// TIA Portal V15.1 export
// export: Created 2024-06-21T08:41:25.9680752Z, ExportSetting WithDefaults, DisplayName Totally Integrated Automation Portal, DisplayVersion V15.1 Update 5, DisplayName TIA Portal Openness, DisplayVersion V15.1 Update 5, DisplayName SINAMICS Startdrive Advanced, DisplayVersion V15.1, DisplayName G130, G150, S120, S150, SINAMICS MV, S210, DisplayVersion V15.1, DisplayName G110M, G120, G120C, G120D, G120P, DisplayVersion V15.1, DisplayName STEP 7 Professional, DisplayVersion V15.1 Update 5, DisplayName STEP 7 Safety, DisplayVersion V15.1, DisplayName WinCC Professional, DisplayVersion V15.1 Update 5, DisplayName SIMATIC Visualization Architect, DisplayVersion V15.1
FUNCTION "209000NCP01EnableAlarms" : Void   // FC198, FBD
TITLE = 209000NCP01EnableAlarms
{ S7_Optimized_Access := 'TRUE' }
VERSION : 0.1
// stored: AutoNumber false, IsIECCheckEnabled false, SetENOAutomatically False, UDAEnableTagReadback false
BEGIN

REGION Network 1: **** --------------------- General --------------------- ****
END_REGION

REGION Network 2: **** 2.1 - Enable Alarms **** General Switch - 209000AE02-JW210
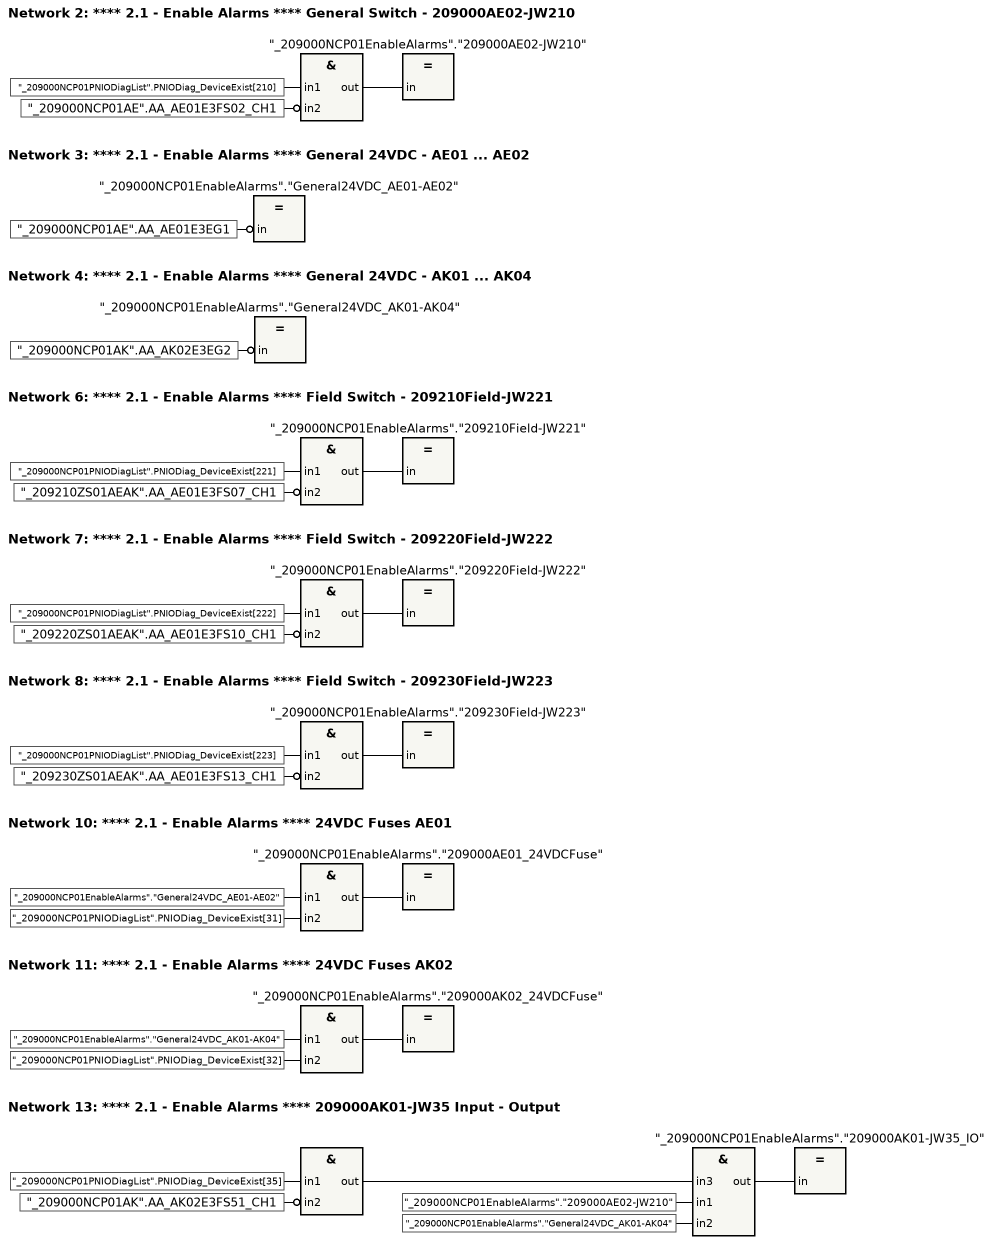
   "_209000NCP01EnableAlarms"."209000AE02-JW210" := "_209000NCP01PNIODiagList".PNIODiag_DeviceExist[210] AND NOT "_209000NCP01AE".AA_AE01E3FS02_CH1;
END_REGION

REGION Network 3: **** 2.1 - Enable Alarms **** General 24VDC - AE01 ... AE02
   "_209000NCP01EnableAlarms"."General24VDC_AE01-AE02" := NOT "_209000NCP01AE".AA_AE01E3EG1;
END_REGION

REGION Network 4: **** 2.1 - Enable Alarms **** General 24VDC - AK01 ... AK04
   "_209000NCP01EnableAlarms"."General24VDC_AK01-AK04" := NOT "_209000NCP01AK".AA_AK02E3EG2;
END_REGION

REGION Network 5: **** --------------------- Field Switch --------------------- ****
END_REGION

REGION Network 6: **** 2.1 - Enable Alarms **** Field Switch - 209210Field-JW221
   "_209000NCP01EnableAlarms"."209210Field-JW221" := "_209000NCP01PNIODiagList".PNIODiag_DeviceExist[221] AND NOT "_209210ZS01AEAK".AA_AE01E3FS07_CH1;
END_REGION

REGION Network 7: **** 2.1 - Enable Alarms **** Field Switch - 209220Field-JW222
   "_209000NCP01EnableAlarms"."209220Field-JW222" := "_209000NCP01PNIODiagList".PNIODiag_DeviceExist[222] AND NOT "_209220ZS01AEAK".AA_AE01E3FS10_CH1;
END_REGION

REGION Network 8: **** 2.1 - Enable Alarms **** Field Switch - 209230Field-JW223
   "_209000NCP01EnableAlarms"."209230Field-JW223" := "_209000NCP01PNIODiagList".PNIODiag_DeviceExist[223] AND NOT "_209230ZS01AEAK".AA_AE01E3FS13_CH1;
END_REGION

REGION Network 9: **** --------------------- ETA Fuse --------------------- ****
END_REGION

REGION Network 10: **** 2.1 - Enable Alarms **** 24VDC Fuses AE01
   "_209000NCP01EnableAlarms"."209000AE01_24VDCFuse" := "_209000NCP01EnableAlarms"."General24VDC_AE01-AE02" AND "_209000NCP01PNIODiagList".PNIODiag_DeviceExist[31];
END_REGION

REGION Network 11: **** 2.1 - Enable Alarms **** 24VDC Fuses AK02
   "_209000NCP01EnableAlarms"."209000AK02_24VDCFuse" := "_209000NCP01EnableAlarms"."General24VDC_AK01-AK04" AND "_209000NCP01PNIODiagList".PNIODiag_DeviceExist[32];
END_REGION

REGION Network 12: **** --------------------- ET200sp I/O --------------------- ****
END_REGION

REGION Network 13: **** 2.1 - Enable Alarms **** 209000AK01-JW35 Input - Output
   "_209000NCP01EnableAlarms"."209000AK01-JW35_IO" := "_209000NCP01PNIODiagList".PNIODiag_DeviceExist[35] AND NOT "_209000NCP01AK".AA_AK02E3FS51_CH1 AND "_209000NCP01EnableAlarms"."209000AE02-JW210" AND "_209000NCP01EnableAlarms"."General24VDC_AK01-AK04";
END_REGION

REGION Network 14: **** 2.1 - Enable Alarms **** 209000AK01-JW35 Safety Input - Output
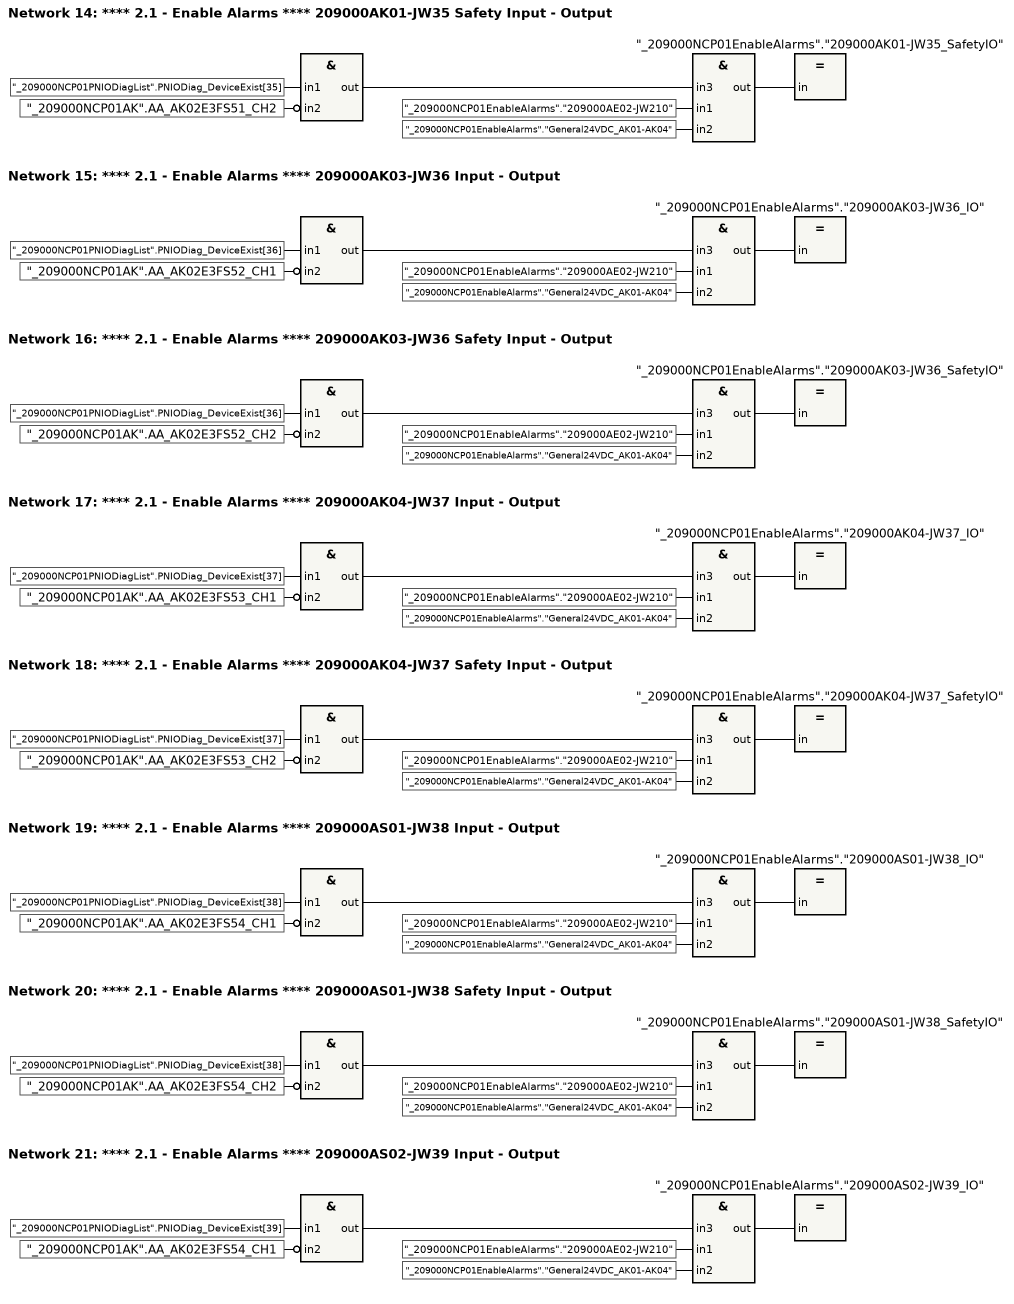
   "_209000NCP01EnableAlarms"."209000AK01-JW35_SafetyIO" := "_209000NCP01PNIODiagList".PNIODiag_DeviceExist[35] AND NOT "_209000NCP01AK".AA_AK02E3FS51_CH2 AND "_209000NCP01EnableAlarms"."209000AE02-JW210" AND "_209000NCP01EnableAlarms"."General24VDC_AK01-AK04";
END_REGION

REGION Network 15: **** 2.1 - Enable Alarms **** 209000AK03-JW36 Input - Output
   "_209000NCP01EnableAlarms"."209000AK03-JW36_IO" := "_209000NCP01PNIODiagList".PNIODiag_DeviceExist[36] AND NOT "_209000NCP01AK".AA_AK02E3FS52_CH1 AND "_209000NCP01EnableAlarms"."209000AE02-JW210" AND "_209000NCP01EnableAlarms"."General24VDC_AK01-AK04";
END_REGION

REGION Network 16: **** 2.1 - Enable Alarms **** 209000AK03-JW36 Safety Input - Output
   "_209000NCP01EnableAlarms"."209000AK03-JW36_SafetyIO" := "_209000NCP01PNIODiagList".PNIODiag_DeviceExist[36] AND NOT "_209000NCP01AK".AA_AK02E3FS52_CH2 AND "_209000NCP01EnableAlarms"."209000AE02-JW210" AND "_209000NCP01EnableAlarms"."General24VDC_AK01-AK04";
END_REGION

REGION Network 17: **** 2.1 - Enable Alarms **** 209000AK04-JW37 Input - Output
   "_209000NCP01EnableAlarms"."209000AK04-JW37_IO" := "_209000NCP01PNIODiagList".PNIODiag_DeviceExist[37] AND NOT "_209000NCP01AK".AA_AK02E3FS53_CH1 AND "_209000NCP01EnableAlarms"."209000AE02-JW210" AND "_209000NCP01EnableAlarms"."General24VDC_AK01-AK04";
END_REGION

REGION Network 18: **** 2.1 - Enable Alarms **** 209000AK04-JW37 Safety Input - Output
   "_209000NCP01EnableAlarms"."209000AK04-JW37_SafetyIO" := "_209000NCP01PNIODiagList".PNIODiag_DeviceExist[37] AND NOT "_209000NCP01AK".AA_AK02E3FS53_CH2 AND "_209000NCP01EnableAlarms"."209000AE02-JW210" AND "_209000NCP01EnableAlarms"."General24VDC_AK01-AK04";
END_REGION

REGION Network 19: **** 2.1 - Enable Alarms **** 209000AS01-JW38 Input - Output
   "_209000NCP01EnableAlarms"."209000AS01-JW38_IO" := "_209000NCP01PNIODiagList".PNIODiag_DeviceExist[38] AND NOT "_209000NCP01AK".AA_AK02E3FS54_CH1 AND "_209000NCP01EnableAlarms"."209000AE02-JW210" AND "_209000NCP01EnableAlarms"."General24VDC_AK01-AK04";
END_REGION

REGION Network 20: **** 2.1 - Enable Alarms **** 209000AS01-JW38 Safety Input - Output
   "_209000NCP01EnableAlarms"."209000AS01-JW38_SafetyIO" := "_209000NCP01PNIODiagList".PNIODiag_DeviceExist[38] AND NOT "_209000NCP01AK".AA_AK02E3FS54_CH2 AND "_209000NCP01EnableAlarms"."209000AE02-JW210" AND "_209000NCP01EnableAlarms"."General24VDC_AK01-AK04";
END_REGION

REGION Network 21: **** 2.1 - Enable Alarms **** 209000AS02-JW39 Input - Output
   "_209000NCP01EnableAlarms"."209000AS02-JW39_IO" := "_209000NCP01PNIODiagList".PNIODiag_DeviceExist[39] AND NOT "_209000NCP01AK".AA_AK02E3FS54_CH1 AND "_209000NCP01EnableAlarms"."209000AE02-JW210" AND "_209000NCP01EnableAlarms"."General24VDC_AK01-AK04";
END_REGION

REGION Network 22: **** 2.1 - Enable Alarms **** 209000AS02-JW39 Safety Input - Output
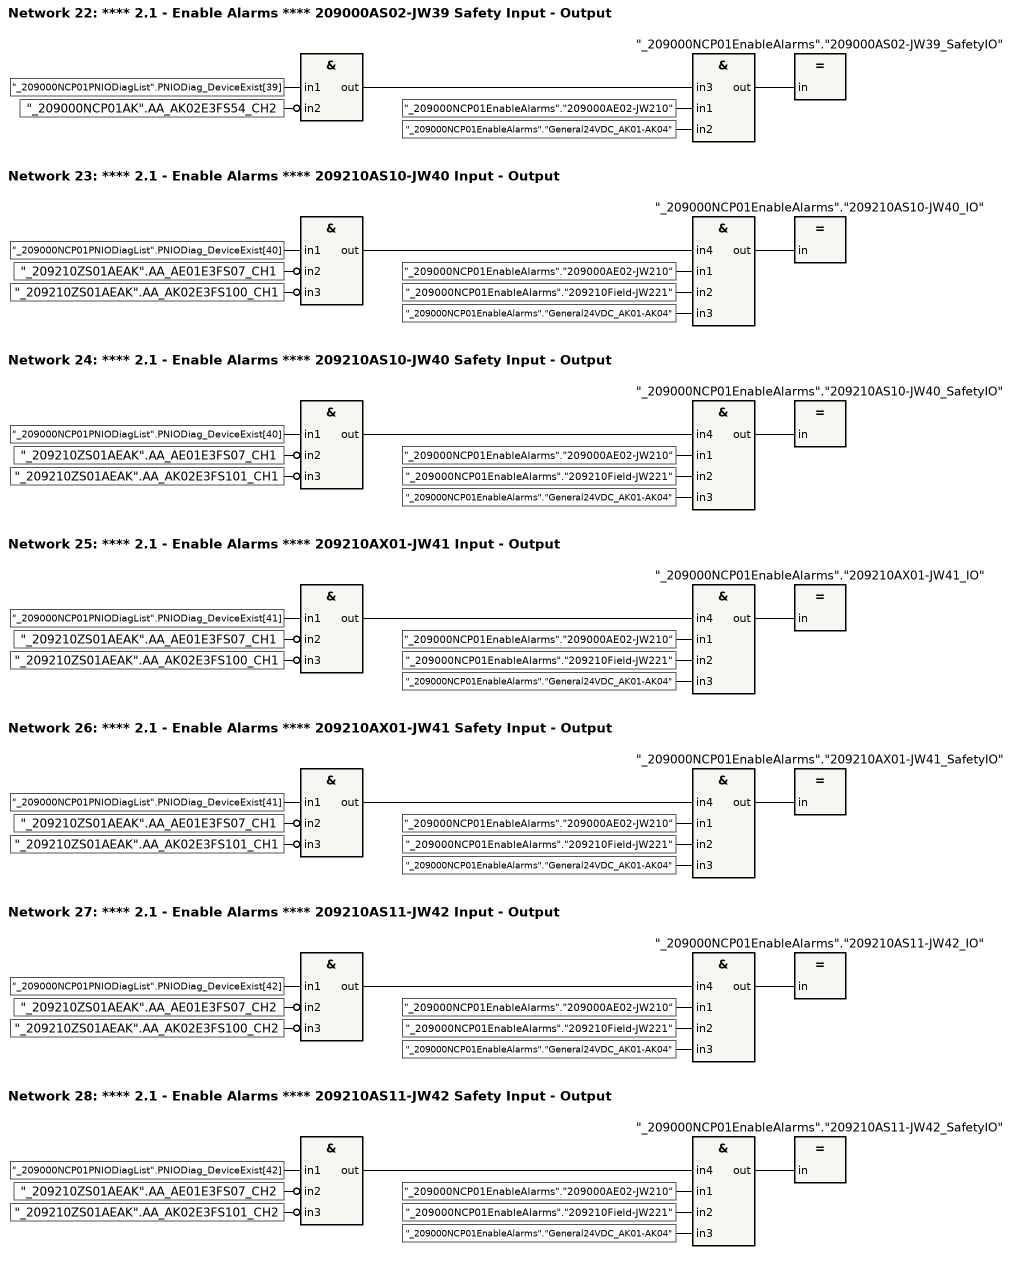
   "_209000NCP01EnableAlarms"."209000AS02-JW39_SafetyIO" := "_209000NCP01PNIODiagList".PNIODiag_DeviceExist[39] AND NOT "_209000NCP01AK".AA_AK02E3FS54_CH2 AND "_209000NCP01EnableAlarms"."209000AE02-JW210" AND "_209000NCP01EnableAlarms"."General24VDC_AK01-AK04";
END_REGION

REGION Network 23: **** 2.1 - Enable Alarms **** 209210AS10-JW40 Input - Output
   "_209000NCP01EnableAlarms"."209210AS10-JW40_IO" := "_209000NCP01PNIODiagList".PNIODiag_DeviceExist[40] AND NOT "_209210ZS01AEAK".AA_AE01E3FS07_CH1 AND NOT "_209210ZS01AEAK".AA_AK02E3FS100_CH1 AND "_209000NCP01EnableAlarms"."209000AE02-JW210" AND "_209000NCP01EnableAlarms"."209210Field-JW221" AND "_209000NCP01EnableAlarms"."General24VDC_AK01-AK04";
END_REGION

REGION Network 24: **** 2.1 - Enable Alarms **** 209210AS10-JW40 Safety Input - Output
   "_209000NCP01EnableAlarms"."209210AS10-JW40_SafetyIO" := "_209000NCP01PNIODiagList".PNIODiag_DeviceExist[40] AND NOT "_209210ZS01AEAK".AA_AE01E3FS07_CH1 AND NOT "_209210ZS01AEAK".AA_AK02E3FS101_CH1 AND "_209000NCP01EnableAlarms"."209000AE02-JW210" AND "_209000NCP01EnableAlarms"."209210Field-JW221" AND "_209000NCP01EnableAlarms"."General24VDC_AK01-AK04";
END_REGION

REGION Network 25: **** 2.1 - Enable Alarms **** 209210AX01-JW41 Input - Output
   "_209000NCP01EnableAlarms"."209210AX01-JW41_IO" := "_209000NCP01PNIODiagList".PNIODiag_DeviceExist[41] AND NOT "_209210ZS01AEAK".AA_AE01E3FS07_CH1 AND NOT "_209210ZS01AEAK".AA_AK02E3FS100_CH1 AND "_209000NCP01EnableAlarms"."209000AE02-JW210" AND "_209000NCP01EnableAlarms"."209210Field-JW221" AND "_209000NCP01EnableAlarms"."General24VDC_AK01-AK04";
END_REGION

REGION Network 26: **** 2.1 - Enable Alarms **** 209210AX01-JW41 Safety Input - Output
   "_209000NCP01EnableAlarms"."209210AX01-JW41_SafetyIO" := "_209000NCP01PNIODiagList".PNIODiag_DeviceExist[41] AND NOT "_209210ZS01AEAK".AA_AE01E3FS07_CH1 AND NOT "_209210ZS01AEAK".AA_AK02E3FS101_CH1 AND "_209000NCP01EnableAlarms"."209000AE02-JW210" AND "_209000NCP01EnableAlarms"."209210Field-JW221" AND "_209000NCP01EnableAlarms"."General24VDC_AK01-AK04";
END_REGION

REGION Network 27: **** 2.1 - Enable Alarms **** 209210AS11-JW42 Input - Output
   "_209000NCP01EnableAlarms"."209210AS11-JW42_IO" := "_209000NCP01PNIODiagList".PNIODiag_DeviceExist[42] AND NOT "_209210ZS01AEAK".AA_AE01E3FS07_CH2 AND NOT "_209210ZS01AEAK".AA_AK02E3FS100_CH2 AND "_209000NCP01EnableAlarms"."209000AE02-JW210" AND "_209000NCP01EnableAlarms"."209210Field-JW221" AND "_209000NCP01EnableAlarms"."General24VDC_AK01-AK04";
END_REGION

REGION Network 28: **** 2.1 - Enable Alarms **** 209210AS11-JW42 Safety Input - Output
   "_209000NCP01EnableAlarms"."209210AS11-JW42_SafetyIO" := "_209000NCP01PNIODiagList".PNIODiag_DeviceExist[42] AND NOT "_209210ZS01AEAK".AA_AE01E3FS07_CH2 AND NOT "_209210ZS01AEAK".AA_AK02E3FS101_CH2 AND "_209000NCP01EnableAlarms"."209000AE02-JW210" AND "_209000NCP01EnableAlarms"."209210Field-JW221" AND "_209000NCP01EnableAlarms"."General24VDC_AK01-AK04";
END_REGION

REGION Network 29: **** 2.1 - Enable Alarms **** 209210AX02-JW43 Input - Output
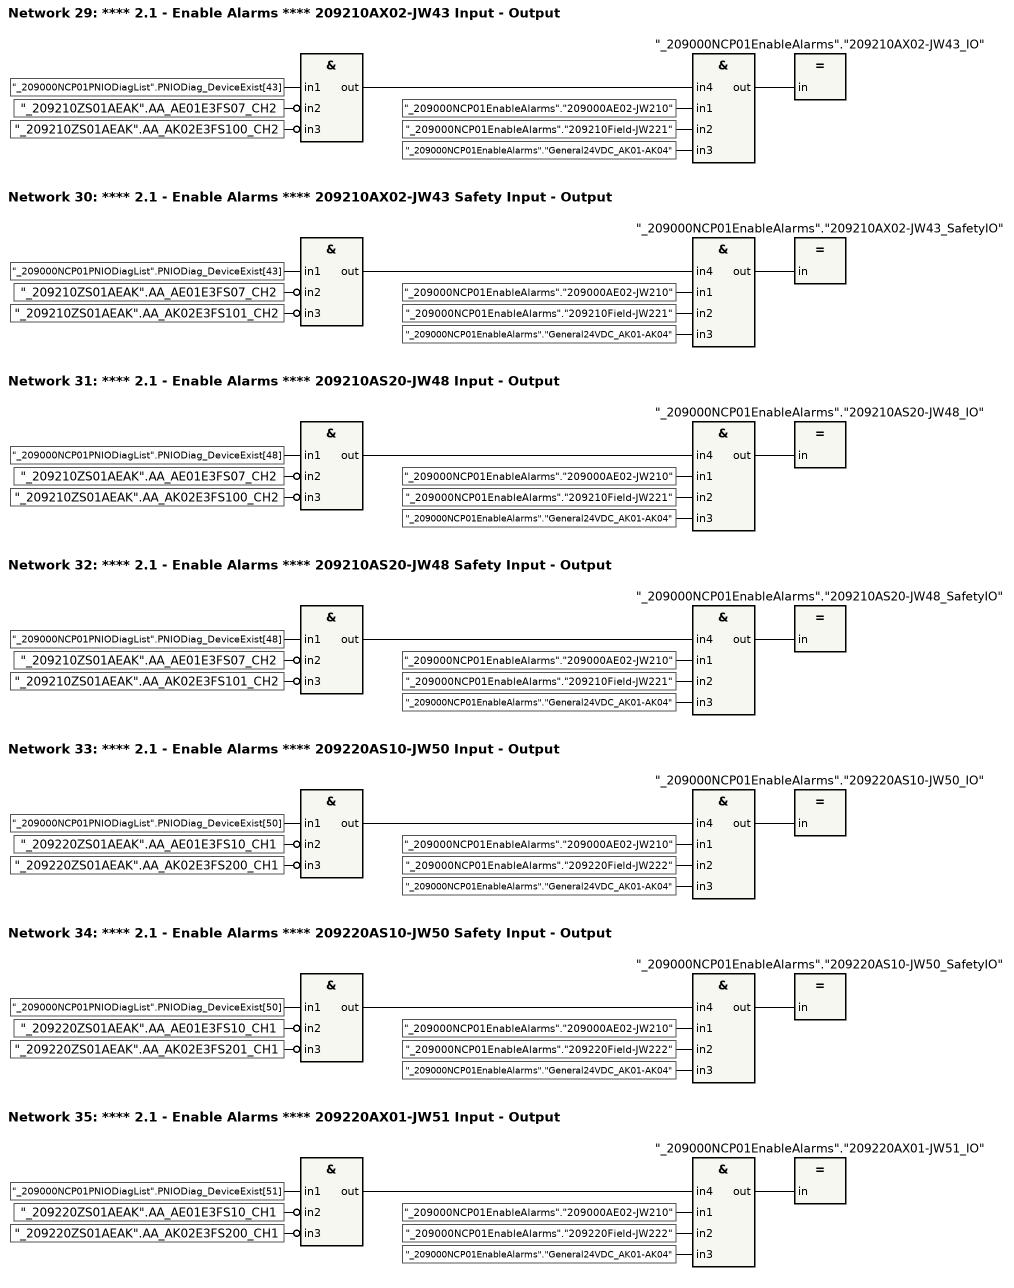
   "_209000NCP01EnableAlarms"."209210AX02-JW43_IO" := "_209000NCP01PNIODiagList".PNIODiag_DeviceExist[43] AND NOT "_209210ZS01AEAK".AA_AE01E3FS07_CH2 AND NOT "_209210ZS01AEAK".AA_AK02E3FS100_CH2 AND "_209000NCP01EnableAlarms"."209000AE02-JW210" AND "_209000NCP01EnableAlarms"."209210Field-JW221" AND "_209000NCP01EnableAlarms"."General24VDC_AK01-AK04";
END_REGION

REGION Network 30: **** 2.1 - Enable Alarms **** 209210AX02-JW43 Safety Input - Output
   "_209000NCP01EnableAlarms"."209210AX02-JW43_SafetyIO" := "_209000NCP01PNIODiagList".PNIODiag_DeviceExist[43] AND NOT "_209210ZS01AEAK".AA_AE01E3FS07_CH2 AND NOT "_209210ZS01AEAK".AA_AK02E3FS101_CH2 AND "_209000NCP01EnableAlarms"."209000AE02-JW210" AND "_209000NCP01EnableAlarms"."209210Field-JW221" AND "_209000NCP01EnableAlarms"."General24VDC_AK01-AK04";
END_REGION

REGION Network 31: **** 2.1 - Enable Alarms **** 209210AS20-JW48 Input - Output
   "_209000NCP01EnableAlarms"."209210AS20-JW48_IO" := "_209000NCP01PNIODiagList".PNIODiag_DeviceExist[48] AND NOT "_209210ZS01AEAK".AA_AE01E3FS07_CH2 AND NOT "_209210ZS01AEAK".AA_AK02E3FS100_CH2 AND "_209000NCP01EnableAlarms"."209000AE02-JW210" AND "_209000NCP01EnableAlarms"."209210Field-JW221" AND "_209000NCP01EnableAlarms"."General24VDC_AK01-AK04";
END_REGION

REGION Network 32: **** 2.1 - Enable Alarms **** 209210AS20-JW48 Safety Input - Output
   "_209000NCP01EnableAlarms"."209210AS20-JW48_SafetyIO" := "_209000NCP01PNIODiagList".PNIODiag_DeviceExist[48] AND NOT "_209210ZS01AEAK".AA_AE01E3FS07_CH2 AND NOT "_209210ZS01AEAK".AA_AK02E3FS101_CH2 AND "_209000NCP01EnableAlarms"."209000AE02-JW210" AND "_209000NCP01EnableAlarms"."209210Field-JW221" AND "_209000NCP01EnableAlarms"."General24VDC_AK01-AK04";
END_REGION

REGION Network 33: **** 2.1 - Enable Alarms **** 209220AS10-JW50 Input - Output
   "_209000NCP01EnableAlarms"."209220AS10-JW50_IO" := "_209000NCP01PNIODiagList".PNIODiag_DeviceExist[50] AND NOT "_209220ZS01AEAK".AA_AE01E3FS10_CH1 AND NOT "_209220ZS01AEAK".AA_AK02E3FS200_CH1 AND "_209000NCP01EnableAlarms"."209000AE02-JW210" AND "_209000NCP01EnableAlarms"."209220Field-JW222" AND "_209000NCP01EnableAlarms"."General24VDC_AK01-AK04";
END_REGION

REGION Network 34: **** 2.1 - Enable Alarms **** 209220AS10-JW50 Safety Input - Output
   "_209000NCP01EnableAlarms"."209220AS10-JW50_SafetyIO" := "_209000NCP01PNIODiagList".PNIODiag_DeviceExist[50] AND NOT "_209220ZS01AEAK".AA_AE01E3FS10_CH1 AND NOT "_209220ZS01AEAK".AA_AK02E3FS201_CH1 AND "_209000NCP01EnableAlarms"."209000AE02-JW210" AND "_209000NCP01EnableAlarms"."209220Field-JW222" AND "_209000NCP01EnableAlarms"."General24VDC_AK01-AK04";
END_REGION

REGION Network 35: **** 2.1 - Enable Alarms **** 209220AX01-JW51 Input - Output
   "_209000NCP01EnableAlarms"."209220AX01-JW51_IO" := "_209000NCP01PNIODiagList".PNIODiag_DeviceExist[51] AND NOT "_209220ZS01AEAK".AA_AE01E3FS10_CH1 AND NOT "_209220ZS01AEAK".AA_AK02E3FS200_CH1 AND "_209000NCP01EnableAlarms"."209000AE02-JW210" AND "_209000NCP01EnableAlarms"."209220Field-JW222" AND "_209000NCP01EnableAlarms"."General24VDC_AK01-AK04";
END_REGION

REGION Network 36: **** 2.1 - Enable Alarms **** 209220AX01-JW51 Safety Input - Output
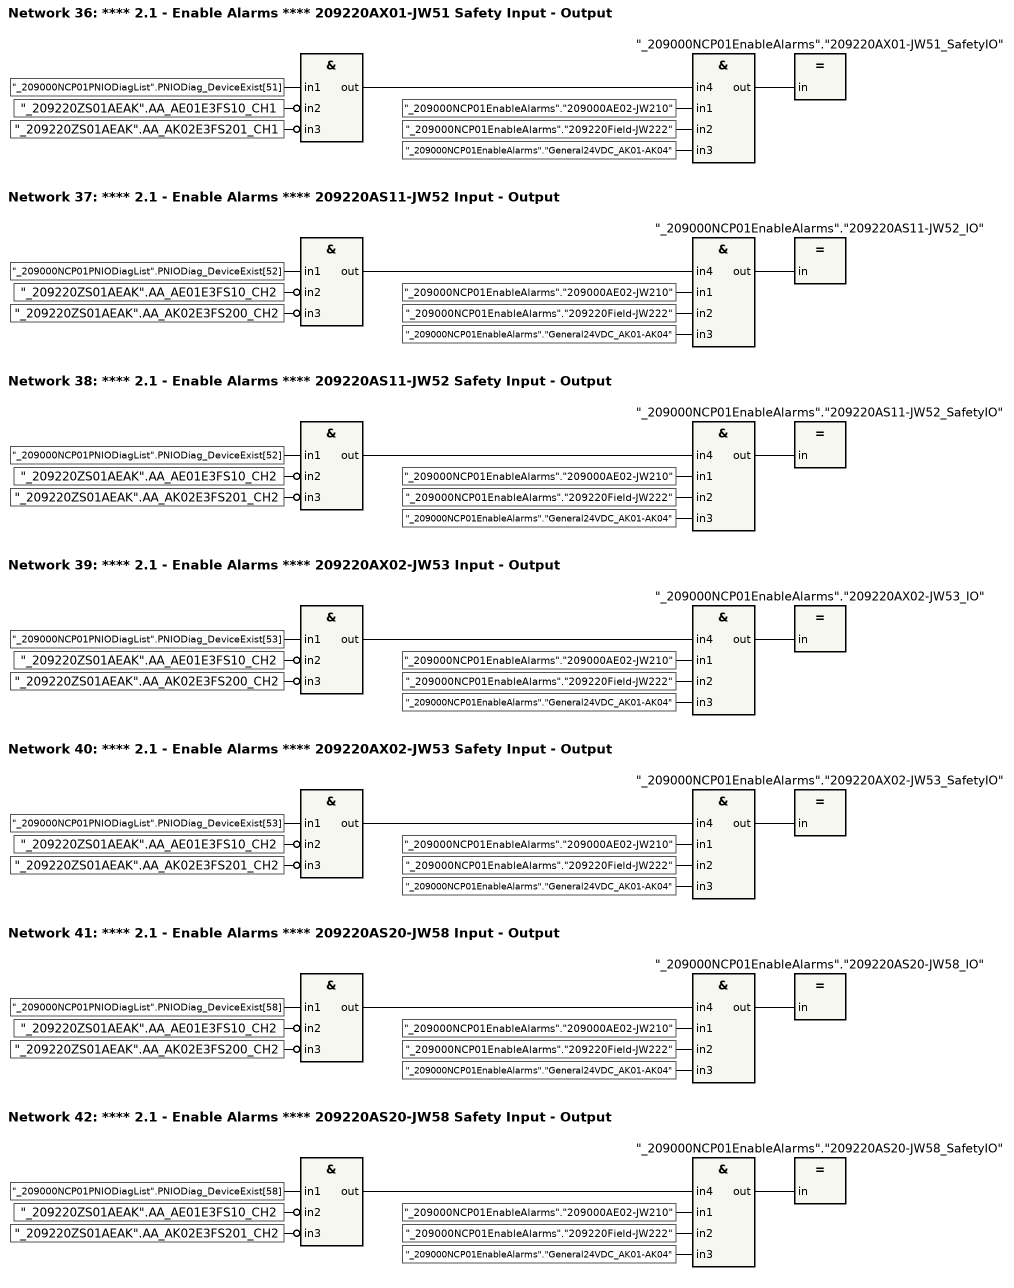
   "_209000NCP01EnableAlarms"."209220AX01-JW51_SafetyIO" := "_209000NCP01PNIODiagList".PNIODiag_DeviceExist[51] AND NOT "_209220ZS01AEAK".AA_AE01E3FS10_CH1 AND NOT "_209220ZS01AEAK".AA_AK02E3FS201_CH1 AND "_209000NCP01EnableAlarms"."209000AE02-JW210" AND "_209000NCP01EnableAlarms"."209220Field-JW222" AND "_209000NCP01EnableAlarms"."General24VDC_AK01-AK04";
END_REGION

REGION Network 37: **** 2.1 - Enable Alarms **** 209220AS11-JW52 Input - Output
   "_209000NCP01EnableAlarms"."209220AS11-JW52_IO" := "_209000NCP01PNIODiagList".PNIODiag_DeviceExist[52] AND NOT "_209220ZS01AEAK".AA_AE01E3FS10_CH2 AND NOT "_209220ZS01AEAK".AA_AK02E3FS200_CH2 AND "_209000NCP01EnableAlarms"."209000AE02-JW210" AND "_209000NCP01EnableAlarms"."209220Field-JW222" AND "_209000NCP01EnableAlarms"."General24VDC_AK01-AK04";
END_REGION

REGION Network 38: **** 2.1 - Enable Alarms **** 209220AS11-JW52 Safety Input - Output
   "_209000NCP01EnableAlarms"."209220AS11-JW52_SafetyIO" := "_209000NCP01PNIODiagList".PNIODiag_DeviceExist[52] AND NOT "_209220ZS01AEAK".AA_AE01E3FS10_CH2 AND NOT "_209220ZS01AEAK".AA_AK02E3FS201_CH2 AND "_209000NCP01EnableAlarms"."209000AE02-JW210" AND "_209000NCP01EnableAlarms"."209220Field-JW222" AND "_209000NCP01EnableAlarms"."General24VDC_AK01-AK04";
END_REGION

REGION Network 39: **** 2.1 - Enable Alarms **** 209220AX02-JW53 Input - Output
   "_209000NCP01EnableAlarms"."209220AX02-JW53_IO" := "_209000NCP01PNIODiagList".PNIODiag_DeviceExist[53] AND NOT "_209220ZS01AEAK".AA_AE01E3FS10_CH2 AND NOT "_209220ZS01AEAK".AA_AK02E3FS200_CH2 AND "_209000NCP01EnableAlarms"."209000AE02-JW210" AND "_209000NCP01EnableAlarms"."209220Field-JW222" AND "_209000NCP01EnableAlarms"."General24VDC_AK01-AK04";
END_REGION

REGION Network 40: **** 2.1 - Enable Alarms **** 209220AX02-JW53 Safety Input - Output
   "_209000NCP01EnableAlarms"."209220AX02-JW53_SafetyIO" := "_209000NCP01PNIODiagList".PNIODiag_DeviceExist[53] AND NOT "_209220ZS01AEAK".AA_AE01E3FS10_CH2 AND NOT "_209220ZS01AEAK".AA_AK02E3FS201_CH2 AND "_209000NCP01EnableAlarms"."209000AE02-JW210" AND "_209000NCP01EnableAlarms"."209220Field-JW222" AND "_209000NCP01EnableAlarms"."General24VDC_AK01-AK04";
END_REGION

REGION Network 41: **** 2.1 - Enable Alarms **** 209220AS20-JW58 Input - Output
   "_209000NCP01EnableAlarms"."209220AS20-JW58_IO" := "_209000NCP01PNIODiagList".PNIODiag_DeviceExist[58] AND NOT "_209220ZS01AEAK".AA_AE01E3FS10_CH2 AND NOT "_209220ZS01AEAK".AA_AK02E3FS200_CH2 AND "_209000NCP01EnableAlarms"."209000AE02-JW210" AND "_209000NCP01EnableAlarms"."209220Field-JW222" AND "_209000NCP01EnableAlarms"."General24VDC_AK01-AK04";
END_REGION

REGION Network 42: **** 2.1 - Enable Alarms **** 209220AS20-JW58 Safety Input - Output
   "_209000NCP01EnableAlarms"."209220AS20-JW58_SafetyIO" := "_209000NCP01PNIODiagList".PNIODiag_DeviceExist[58] AND NOT "_209220ZS01AEAK".AA_AE01E3FS10_CH2 AND NOT "_209220ZS01AEAK".AA_AK02E3FS201_CH2 AND "_209000NCP01EnableAlarms"."209000AE02-JW210" AND "_209000NCP01EnableAlarms"."209220Field-JW222" AND "_209000NCP01EnableAlarms"."General24VDC_AK01-AK04";
END_REGION

REGION Network 43: **** 2.1 - Enable Alarms **** 209230AS10-JW60 Input - Output
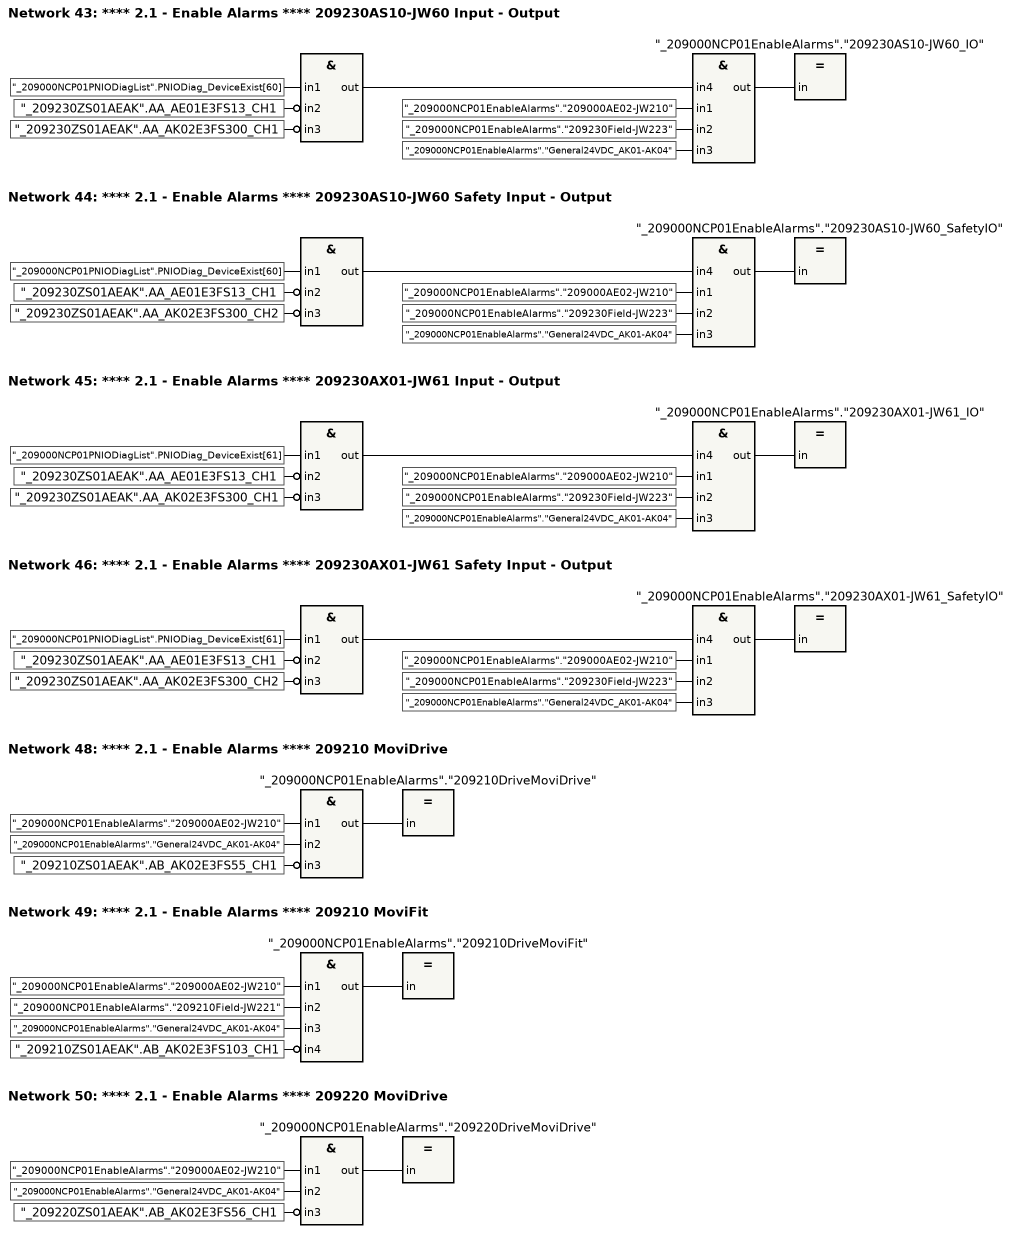
   "_209000NCP01EnableAlarms"."209230AS10-JW60_IO" := "_209000NCP01PNIODiagList".PNIODiag_DeviceExist[60] AND NOT "_209230ZS01AEAK".AA_AE01E3FS13_CH1 AND NOT "_209230ZS01AEAK".AA_AK02E3FS300_CH1 AND "_209000NCP01EnableAlarms"."209000AE02-JW210" AND "_209000NCP01EnableAlarms"."209230Field-JW223" AND "_209000NCP01EnableAlarms"."General24VDC_AK01-AK04";
END_REGION

REGION Network 44: **** 2.1 - Enable Alarms **** 209230AS10-JW60 Safety Input - Output
   "_209000NCP01EnableAlarms"."209230AS10-JW60_SafetyIO" := "_209000NCP01PNIODiagList".PNIODiag_DeviceExist[60] AND NOT "_209230ZS01AEAK".AA_AE01E3FS13_CH1 AND NOT "_209230ZS01AEAK".AA_AK02E3FS300_CH2 AND "_209000NCP01EnableAlarms"."209000AE02-JW210" AND "_209000NCP01EnableAlarms"."209230Field-JW223" AND "_209000NCP01EnableAlarms"."General24VDC_AK01-AK04";
END_REGION

REGION Network 45: **** 2.1 - Enable Alarms **** 209230AX01-JW61 Input - Output
   "_209000NCP01EnableAlarms"."209230AX01-JW61_IO" := "_209000NCP01PNIODiagList".PNIODiag_DeviceExist[61] AND NOT "_209230ZS01AEAK".AA_AE01E3FS13_CH1 AND NOT "_209230ZS01AEAK".AA_AK02E3FS300_CH1 AND "_209000NCP01EnableAlarms"."209000AE02-JW210" AND "_209000NCP01EnableAlarms"."209230Field-JW223" AND "_209000NCP01EnableAlarms"."General24VDC_AK01-AK04";
END_REGION

REGION Network 46: **** 2.1 - Enable Alarms **** 209230AX01-JW61 Safety Input - Output
   "_209000NCP01EnableAlarms"."209230AX01-JW61_SafetyIO" := "_209000NCP01PNIODiagList".PNIODiag_DeviceExist[61] AND NOT "_209230ZS01AEAK".AA_AE01E3FS13_CH1 AND NOT "_209230ZS01AEAK".AA_AK02E3FS300_CH2 AND "_209000NCP01EnableAlarms"."209000AE02-JW210" AND "_209000NCP01EnableAlarms"."209230Field-JW223" AND "_209000NCP01EnableAlarms"."General24VDC_AK01-AK04";
END_REGION

REGION Network 47: **** --------------------- Drives --------------------- ****
END_REGION

REGION Network 48: **** 2.1 - Enable Alarms **** 209210 MoviDrive
   "_209000NCP01EnableAlarms"."209210DriveMoviDrive" := "_209000NCP01EnableAlarms"."209000AE02-JW210" AND "_209000NCP01EnableAlarms"."General24VDC_AK01-AK04" AND NOT "_209210ZS01AEAK".AB_AK02E3FS55_CH1;
END_REGION

REGION Network 49: **** 2.1 - Enable Alarms **** 209210 MoviFit
   "_209000NCP01EnableAlarms"."209210DriveMoviFit" := "_209000NCP01EnableAlarms"."209000AE02-JW210" AND "_209000NCP01EnableAlarms"."209210Field-JW221" AND "_209000NCP01EnableAlarms"."General24VDC_AK01-AK04" AND NOT "_209210ZS01AEAK".AB_AK02E3FS103_CH1;
END_REGION

REGION Network 50: **** 2.1 - Enable Alarms **** 209220 MoviDrive
   "_209000NCP01EnableAlarms"."209220DriveMoviDrive" := "_209000NCP01EnableAlarms"."209000AE02-JW210" AND "_209000NCP01EnableAlarms"."General24VDC_AK01-AK04" AND NOT "_209220ZS01AEAK".AB_AK02E3FS56_CH1;
END_REGION

REGION Network 51: **** 2.1 - Enable Alarms **** 209220 MoviFit
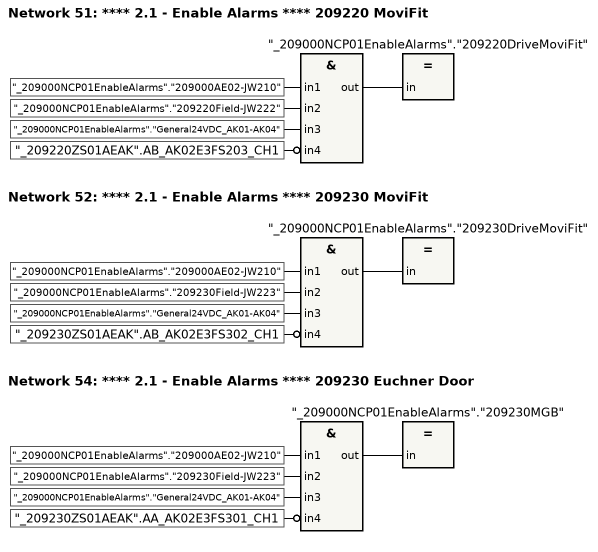
   "_209000NCP01EnableAlarms"."209220DriveMoviFit" := "_209000NCP01EnableAlarms"."209000AE02-JW210" AND "_209000NCP01EnableAlarms"."209220Field-JW222" AND "_209000NCP01EnableAlarms"."General24VDC_AK01-AK04" AND NOT "_209220ZS01AEAK".AB_AK02E3FS203_CH1;
END_REGION

REGION Network 52: **** 2.1 - Enable Alarms **** 209230 MoviFit
   "_209000NCP01EnableAlarms"."209230DriveMoviFit" := "_209000NCP01EnableAlarms"."209000AE02-JW210" AND "_209000NCP01EnableAlarms"."209230Field-JW223" AND "_209000NCP01EnableAlarms"."General24VDC_AK01-AK04" AND NOT "_209230ZS01AEAK".AB_AK02E3FS302_CH1;
END_REGION

REGION Network 53: **** --------------------- Euchner Door --------------------- ****
END_REGION

REGION Network 54: **** 2.1 - Enable Alarms **** 209230 Euchner Door
   "_209000NCP01EnableAlarms"."209230MGB" := "_209000NCP01EnableAlarms"."209000AE02-JW210" AND "_209000NCP01EnableAlarms"."209230Field-JW223" AND "_209000NCP01EnableAlarms"."General24VDC_AK01-AK04" AND NOT "_209230ZS01AEAK".AA_AK02E3FS301_CH1;
END_REGION
END_FUNCTION
